// TIA Portal V20 export
FUNCTION_BLOCK "zGM SafetyGlobalChecksum"   // FB5710, LAD
TITLE = GM Drive Safety Global Checksum
AUTHOR : TayNara
FAMILY : GM_CITI_3_2
VERSION : 1.0
// This logic is for combining parameter 9781[0] of each Control Unit Track changes of Safety functionality  checksums and PLC Safety Signature checksum to create a global single Safety Checksum for the machine. This logic is for auditing purposes and is not considered safety listed or protected use at own risk.
// stored: MemoryReserve 100, SetENOAutomatically false
   VAR_INPUT
      Start : Bool;   // First scan bit.
      ReadFrequency : Time;   // Set time to update the single checksum.
      HardwareID_CU1 : HW_IO;   // Control Unit hardware ID.
      HardwareID_CU2 : HW_IO;   // Control Unit hardware ID.
      HardwareID_CU3 : HW_IO;   // Control Unit hardware ID.
      HardwareID_CU4 : HW_IO;   // Control Unit hardware ID.
      HardwareID_CU5 : HW_IO;   // Control Unit hardware ID.
      HardwareID_CU6 : HW_IO;   // Control Unit hardware ID.
      PlcSafetySignatureIn : DWord;   // PLC Safety Signature from F_SystemInfo_DB.
   END_VAR
   VAR_OUTPUT
      SingleSafetyChecksum : DWord;   // Global Single Safety Signature checksum.
      Busy : Bool;
      Error : Bool;
   END_VAR
   VAR
      instSinaParaS { S7_SetPoint := 'True'} : Array[1..6] of SinaParaS;
      statEnableReadSeq : Bool;   // Enable read sequence.
      statStartFN : Bool;   // Start combining Xor checksums on negative trigger.
      statFreqTimer1 { S7_SetPoint := 'True'} : TON_TIME;
      statFreqTimer2 { S7_SetPoint := 'True'} : TON_TIME;
      statSafetyChecksum { S7_SetPoint := 'True'} : DWord;
      statTimeUp { S7_SetPoint := 'True'} : Bool;
      statTimeUpFP : Bool;
      statReadFrequency : Time;
      statResetEnableFP : Bool;
   END_VAR
   VAR CONSTANT
      CU_SAFETYCHKSUM_PAR_NR : UInt := 9781;   // CU Paramter 9781[0] SI Checksum to track functional changes
   END_VAR
   VAR_TEMP   // added for the SCL form of the ladder/FBD networks
      _w1 : Bool;
      _w2 : Bool;
   END_VAR
BEGIN

REGION Network 1: Preventing read frequency to be set below 30 seconds and moving read frequency time to timer logic
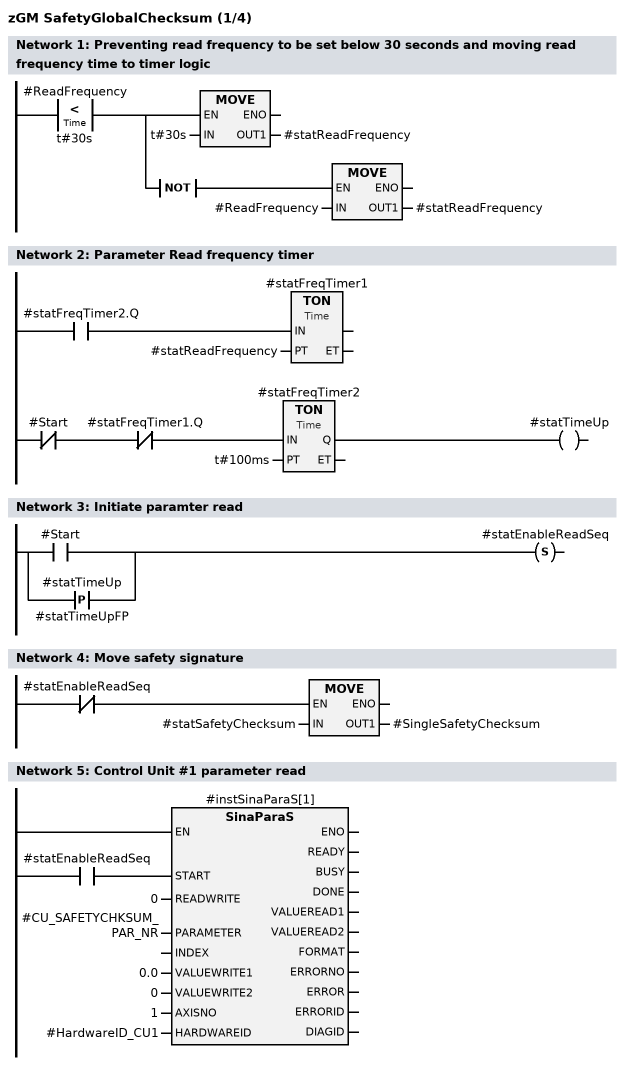
   RUNG wire#powerrail
      { S7_Templates := "SrcType := Time" } LT_Contact(in1 := #ReadFrequency, in2 := t#30s)
      wire#w1
      Move(in := t#30s, out1 => #statReadFrequency)
   END_RUNG
   RUNG wire#w1
      Not()
      Move(in := #ReadFrequency, out1 => #statReadFrequency)
   END_RUNG
   // the same network as SCL:
   #_w1 := #ReadFrequency < t#30s;
   IF #_w1 THEN #statReadFrequency := t#30s; END_IF;
   IF NOT #_w1 THEN #statReadFrequency := #ReadFrequency; END_IF;
END_REGION

REGION Network 2: Parameter Read frequency timer
   RUNG wire#powerrail
      Contact( #statFreqTimer2.Q )
      { S7_Templates := "time_type := Time" } #statFreqTimer1.TON(pt := #statReadFrequency, et =>)
   END_RUNG
   RUNG wire#powerrail
      I_Contact( #Start )
      I_Contact( #statFreqTimer1.Q )
      { S7_Templates := "time_type := Time" } #statFreqTimer2.TON(pt := t#100ms, et =>)
      Coil( #statTimeUp )
   END_RUNG
   // the same network as SCL:
   #statFreqTimer1(IN := #statFreqTimer2.Q, PT := #statReadFrequency);   // TON
   #statFreqTimer2(IN := NOT #Start AND NOT #statFreqTimer1.Q, PT := t#100ms);   // TON
   #statTimeUp := #statFreqTimer2.Q;
END_REGION

REGION Network 3: Initiate paramter read
   RUNG wire#powerrail
      Contact( #Start )
      wire#w1
      S_Coil( #statEnableReadSeq )
   END_RUNG
   RUNG wire#powerrail
      P_Contact(operand := #statTimeUp, bit := #statTimeUpFP)
   END_RUNG wire#w1
   // the same network as SCL:
   #_w1 := #statTimeUp AND NOT #statTimeUpFP;   // rising edge of #statTimeUp
   #statTimeUpFP := #statTimeUp;
   IF #Start OR #_w1 THEN #statEnableReadSeq := TRUE; END_IF;
END_REGION

REGION Network 4: Move safety signature
   RUNG wire#powerrail
      I_Contact( #statEnableReadSeq )
      Move(in := #statSafetyChecksum, out1 => #SingleSafetyChecksum)
   END_RUNG
   // the same network as SCL:
   IF NOT #statEnableReadSeq THEN #SingleSafetyChecksum := #statSafetyChecksum; END_IF;
END_REGION

REGION Network 5: Control Unit #1 parameter read
   RUNG wire#powerrail
      #instSinaParaS[1].SinaParaS(Start := wire#w1, ReadWrite := 0, Parameter := #CU_SAFETYCHKSUM_PAR_NR, Index :=, ValueWrite1 := 0.0, ValueWrite2 := 0, AxisNo := 1, hardwareId := #HardwareID_CU1, Ready =>, Busy =>, Done =>, ValueRead1 =>, ValueRead2 =>, Format =>, ErrorNo =>, Error =>, ErrorId =>, DiagId =>)
   END_RUNG
   RUNG wire#powerrail
      Contact( #statEnableReadSeq )
   END_RUNG wire#w1
   // the same network as SCL:
   #instSinaParaS[1](Start := #statEnableReadSeq,   // SinaParaS
                     ReadWrite := 0,
                     Parameter := #CU_SAFETYCHKSUM_PAR_NR,
                     ValueWrite1 := 0.0,
                     ValueWrite2 := 0,
                     AxisNo := 1,
                     hardwareId := #HardwareID_CU1);
END_REGION

REGION Network 6: Control Unit #2 parameter read
   // #statGetChksum[2]
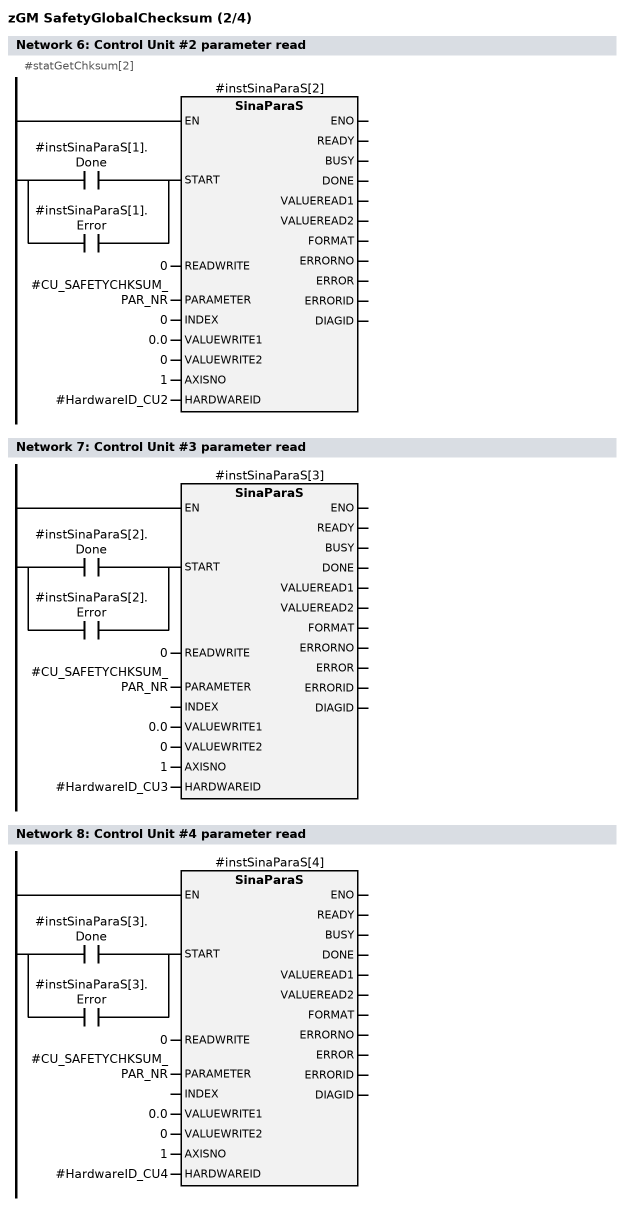
   RUNG wire#powerrail
      #instSinaParaS[2].SinaParaS(Start := wire#w1, ReadWrite := 0, Parameter := #CU_SAFETYCHKSUM_PAR_NR, Index := 0, ValueWrite1 := 0.0, ValueWrite2 := 0, AxisNo := 1, hardwareId := #HardwareID_CU2, Ready =>, Busy =>, Done =>, ValueRead1 =>, ValueRead2 =>, Format =>, ErrorNo =>, Error =>, ErrorId =>, DiagId =>)
   END_RUNG
   RUNG wire#powerrail
      Contact( #instSinaParaS[1].Done )
   END_RUNG wire#w1
   RUNG wire#powerrail
      Contact( #instSinaParaS[1].Error )
   END_RUNG wire#w1
   // the same network as SCL:
   #instSinaParaS[2](Start := #instSinaParaS[1].Done OR #instSinaParaS[1].Error,   // SinaParaS
                     ReadWrite := 0,
                     Parameter := #CU_SAFETYCHKSUM_PAR_NR,
                     Index := 0,
                     ValueWrite1 := 0.0,
                     ValueWrite2 := 0,
                     AxisNo := 1,
                     hardwareId := #HardwareID_CU2);
END_REGION

REGION Network 7: Control Unit #3 parameter read
   RUNG wire#powerrail
      #instSinaParaS[3].SinaParaS(Start := wire#w1, ReadWrite := 0, Parameter := #CU_SAFETYCHKSUM_PAR_NR, Index :=, ValueWrite1 := 0.0, ValueWrite2 := 0, AxisNo := 1, hardwareId := #HardwareID_CU3, Ready =>, Busy =>, Done =>, ValueRead1 =>, ValueRead2 =>, Format =>, ErrorNo =>, Error =>, ErrorId =>, DiagId =>)
   END_RUNG
   RUNG wire#powerrail
      Contact( #instSinaParaS[2].Done )
   END_RUNG wire#w1
   RUNG wire#powerrail
      Contact( #instSinaParaS[2].Error )
   END_RUNG wire#w1
   // the same network as SCL:
   #instSinaParaS[3](Start := #instSinaParaS[2].Done OR #instSinaParaS[2].Error,   // SinaParaS
                     ReadWrite := 0,
                     Parameter := #CU_SAFETYCHKSUM_PAR_NR,
                     ValueWrite1 := 0.0,
                     ValueWrite2 := 0,
                     AxisNo := 1,
                     hardwareId := #HardwareID_CU3);
END_REGION

REGION Network 8: Control Unit #4 parameter read
   RUNG wire#powerrail
      #instSinaParaS[4].SinaParaS(Start := wire#w1, ReadWrite := 0, Parameter := #CU_SAFETYCHKSUM_PAR_NR, Index :=, ValueWrite1 := 0.0, ValueWrite2 := 0, AxisNo := 1, hardwareId := #HardwareID_CU4, Ready =>, Busy =>, Done =>, ValueRead1 =>, ValueRead2 =>, Format =>, ErrorNo =>, Error =>, ErrorId =>, DiagId =>)
   END_RUNG
   RUNG wire#powerrail
      Contact( #instSinaParaS[3].Done )
   END_RUNG wire#w1
   RUNG wire#powerrail
      Contact( #instSinaParaS[3].Error )
   END_RUNG wire#w1
   // the same network as SCL:
   #instSinaParaS[4](Start := #instSinaParaS[3].Done OR #instSinaParaS[3].Error,   // SinaParaS
                     ReadWrite := 0,
                     Parameter := #CU_SAFETYCHKSUM_PAR_NR,
                     ValueWrite1 := 0.0,
                     ValueWrite2 := 0,
                     AxisNo := 1,
                     hardwareId := #HardwareID_CU4);
END_REGION

REGION Network 9: Control Unit #5 parameter read
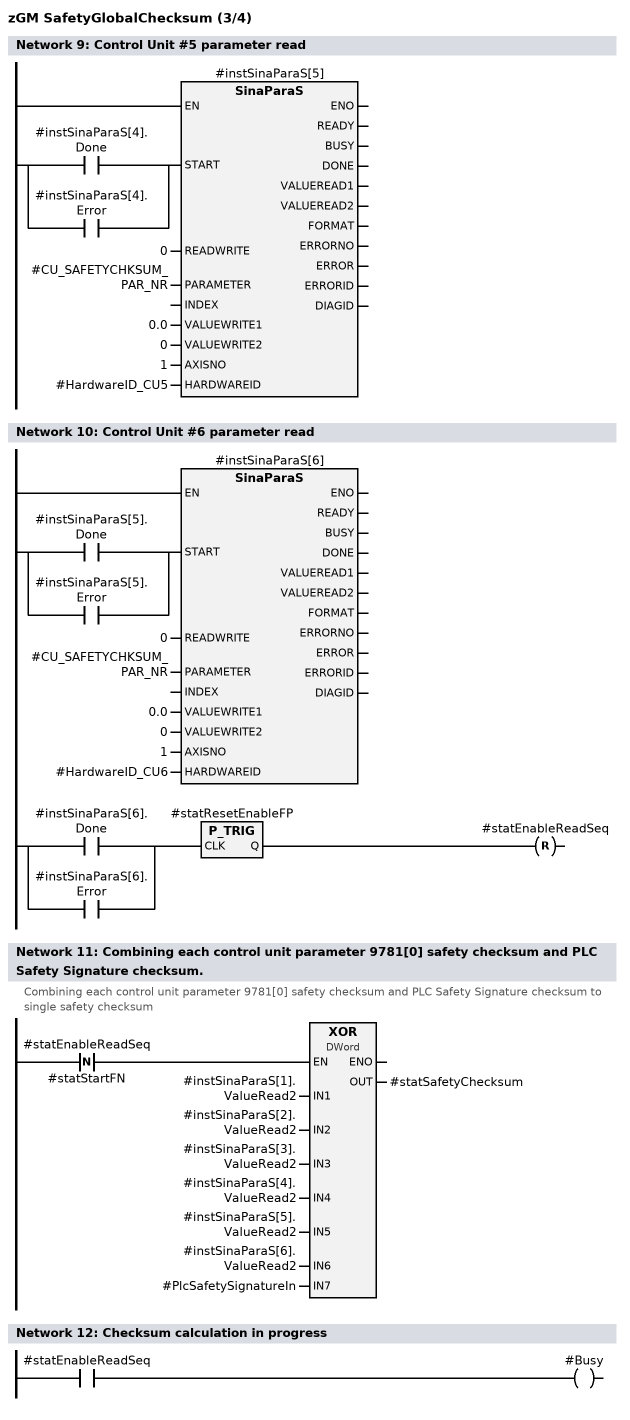
   RUNG wire#powerrail
      #instSinaParaS[5].SinaParaS(Start := wire#w1, ReadWrite := 0, Parameter := #CU_SAFETYCHKSUM_PAR_NR, Index :=, ValueWrite1 := 0.0, ValueWrite2 := 0, AxisNo := 1, hardwareId := #HardwareID_CU5, Ready =>, Busy =>, Done =>, ValueRead1 =>, ValueRead2 =>, Format =>, ErrorNo =>, Error =>, ErrorId =>, DiagId =>)
   END_RUNG
   RUNG wire#powerrail
      Contact( #instSinaParaS[4].Done )
   END_RUNG wire#w1
   RUNG wire#powerrail
      Contact( #instSinaParaS[4].Error )
   END_RUNG wire#w1
   // the same network as SCL:
   #instSinaParaS[5](Start := #instSinaParaS[4].Done OR #instSinaParaS[4].Error,   // SinaParaS
                     ReadWrite := 0,
                     Parameter := #CU_SAFETYCHKSUM_PAR_NR,
                     ValueWrite1 := 0.0,
                     ValueWrite2 := 0,
                     AxisNo := 1,
                     hardwareId := #HardwareID_CU5);
END_REGION

REGION Network 10: Control Unit #6 parameter read
   RUNG wire#powerrail
      #instSinaParaS[6].SinaParaS(Start := wire#w1, ReadWrite := 0, Parameter := #CU_SAFETYCHKSUM_PAR_NR, Index :=, ValueWrite1 := 0.0, ValueWrite2 := 0, AxisNo := 1, hardwareId := #HardwareID_CU6, Ready =>, Busy =>, Done =>, ValueRead1 =>, ValueRead2 =>, Format =>, ErrorNo =>, Error =>, ErrorId =>, DiagId =>)
   END_RUNG
   RUNG wire#powerrail
      Contact( #instSinaParaS[5].Done )
   END_RUNG wire#w1
   RUNG wire#powerrail
      Contact( #instSinaParaS[5].Error )
   END_RUNG wire#w1
   RUNG wire#powerrail
      Contact( #instSinaParaS[6].Done )
      wire#w2
      P_Trig( #statResetEnableFP )
      R_Coil( #statEnableReadSeq )
   END_RUNG
   RUNG wire#powerrail
      Contact( #instSinaParaS[6].Error )
   END_RUNG wire#w2
   // the same network as SCL:
   #instSinaParaS[6](Start := #instSinaParaS[5].Done OR #instSinaParaS[5].Error,   // SinaParaS
                     ReadWrite := 0,
                     Parameter := #CU_SAFETYCHKSUM_PAR_NR,
                     ValueWrite1 := 0.0,
                     ValueWrite2 := 0,
                     AxisNo := 1,
                     hardwareId := #HardwareID_CU6);
   #_w1 := #instSinaParaS[6].Done OR #instSinaParaS[6].Error;
   #_w2 := #_w1 AND NOT #statResetEnableFP;   // rising edge
   #statResetEnableFP := #_w1;
   IF #_w2 THEN #statEnableReadSeq := FALSE; END_IF;
END_REGION

REGION Network 11: Combining each control unit parameter 9781[0] safety checksum and PLC Safety Signature checksum.
   // Combining each control unit parameter 9781[0] safety checksum and PLC Safety Signature checksum to single safety checksum
   #_w1 := NOT #statEnableReadSeq AND #statStartFN;   // falling edge of #statEnableReadSeq
   #statStartFN := #statEnableReadSeq;
   IF #_w1 THEN
       #statSafetyChecksum := #instSinaParaS[1].ValueRead2 XOR #instSinaParaS[2].ValueRead2 XOR #instSinaParaS[3].ValueRead2 XOR #instSinaParaS[4].ValueRead2 XOR #instSinaParaS[5].ValueRead2 XOR #instSinaParaS[6].ValueRead2 XOR #PlcSafetySignatureIn;
   END_IF;
END_REGION

REGION Network 12: Checksum calculation in progress
   RUNG wire#powerrail
      Contact( #statEnableReadSeq )
      Coil( #Busy )
   END_RUNG
   // the same network as SCL:
   #Busy := #statEnableReadSeq;
END_REGION

REGION Network 13: Output error from SINAPARAS read block
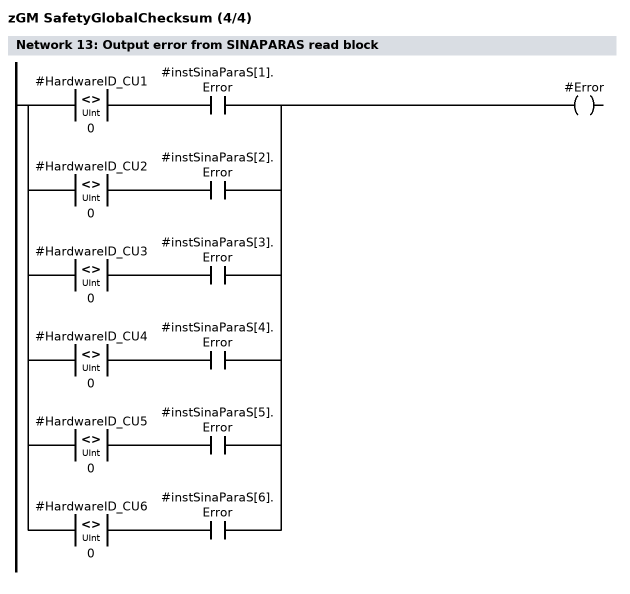
   RUNG wire#powerrail
      { S7_Templates := "SrcType := UInt" } NE_Contact(in1 := #HardwareID_CU1, in2 := 0)
      Contact( #instSinaParaS[1].Error )
      wire#w1
      Coil( #Error )
   END_RUNG
   RUNG wire#powerrail
      { S7_Templates := "SrcType := UInt" } NE_Contact(in1 := #HardwareID_CU2, in2 := 0)
      Contact( #instSinaParaS[2].Error )
   END_RUNG wire#w1
   RUNG wire#powerrail
      { S7_Templates := "SrcType := UInt" } NE_Contact(in1 := #HardwareID_CU3, in2 := 0)
      Contact( #instSinaParaS[3].Error )
   END_RUNG wire#w1
   RUNG wire#powerrail
      { S7_Templates := "SrcType := UInt" } NE_Contact(in1 := #HardwareID_CU4, in2 := 0)
      Contact( #instSinaParaS[4].Error )
   END_RUNG wire#w1
   RUNG wire#powerrail
      { S7_Templates := "SrcType := UInt" } NE_Contact(in1 := #HardwareID_CU5, in2 := 0)
      Contact( #instSinaParaS[5].Error )
   END_RUNG wire#w1
   RUNG wire#powerrail
      { S7_Templates := "SrcType := UInt" } NE_Contact(in1 := #HardwareID_CU6, in2 := 0)
      Contact( #instSinaParaS[6].Error )
   END_RUNG wire#w1
   // the same network as SCL:
   #Error := ((#HardwareID_CU1 <> 0) AND #instSinaParaS[1].Error) OR ((#HardwareID_CU2 <> 0) AND #instSinaParaS[2].Error) OR ((#HardwareID_CU3 <> 0) AND #instSinaParaS[3].Error) OR ((#HardwareID_CU4 <> 0) AND #instSinaParaS[4].Error) OR ((#HardwareID_CU5 <> 0) AND #instSinaParaS[5].Error) OR ((#HardwareID_CU6 <> 0) AND #instSinaParaS[6].Error);
END_REGION
END_FUNCTION_BLOCK
